// Mitsubishi GX Works2 project: Pract03_- Timer01   PLC: FX3U/FX3UC

PROGRAM MAIN
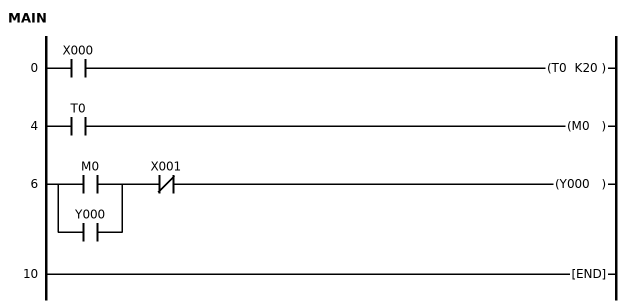
0     LD      X000
      OUT     T0 K20
4     LD      T0
      OUT     M0
6     LD      M0
      OR      Y000
      ANI     X001
      OUT     Y000
10    END
END_PROGRAM
